INTERFACE I_Chain

PROPERTY getDefinition : ST_ChainDefinition
GET
END_GET
END_PROPERTY

PROPERTY getRefChainReleases : REFERENCE TO ARRAY[1..cMaxChains] OF BOOL
GET
END_GET
END_PROPERTY

PROPERTY getRefReleaseResult : REFERENCE TO BOOL
GET
END_GET
END_PROPERTY

END_INTERFACE

(* stored: Version 1.1.0.1, ProductVersion 3.1.4024.0
   Itf I_Chain: Id {7715b3d1-50ff-4b92-8bb5-0e96c4e05098}
   Property getDefinition: Id {ddc1d10c-6789-4589-b30f-51edf9a15f33}
   Get Get: Id {d489da7f-1a23-4aa9-91d4-d2d9d7dca888}
   Property getRefChainReleases: Id {e5db7089-1d60-4597-8d73-a70758c50743}
   Get Get: Id {0292425b-d1ca-42b1-af29-8119aee9f933}
   Property getRefReleaseResult: Id {b5b91659-716c-4627-9804-1bb171c9d22f}
   Get Get: Id {6f931fb6-d496-4f01-aa15-3441af1f65c3} *)
